{attribute 'qualified_only'}
VAR_GLOBAL
		EtherCAT_Master_EJxxxx : EtherCAT_Master_EJxxxx_6E0B2FA6;
END_VAR

(* stored: Version 1.2.0.0, ProductVersion 3.1.4024.9
   GVL GVL_iXlinker: Id {0ca71c5a-a50c-4e55-9213-09f83b76f33d} *)
